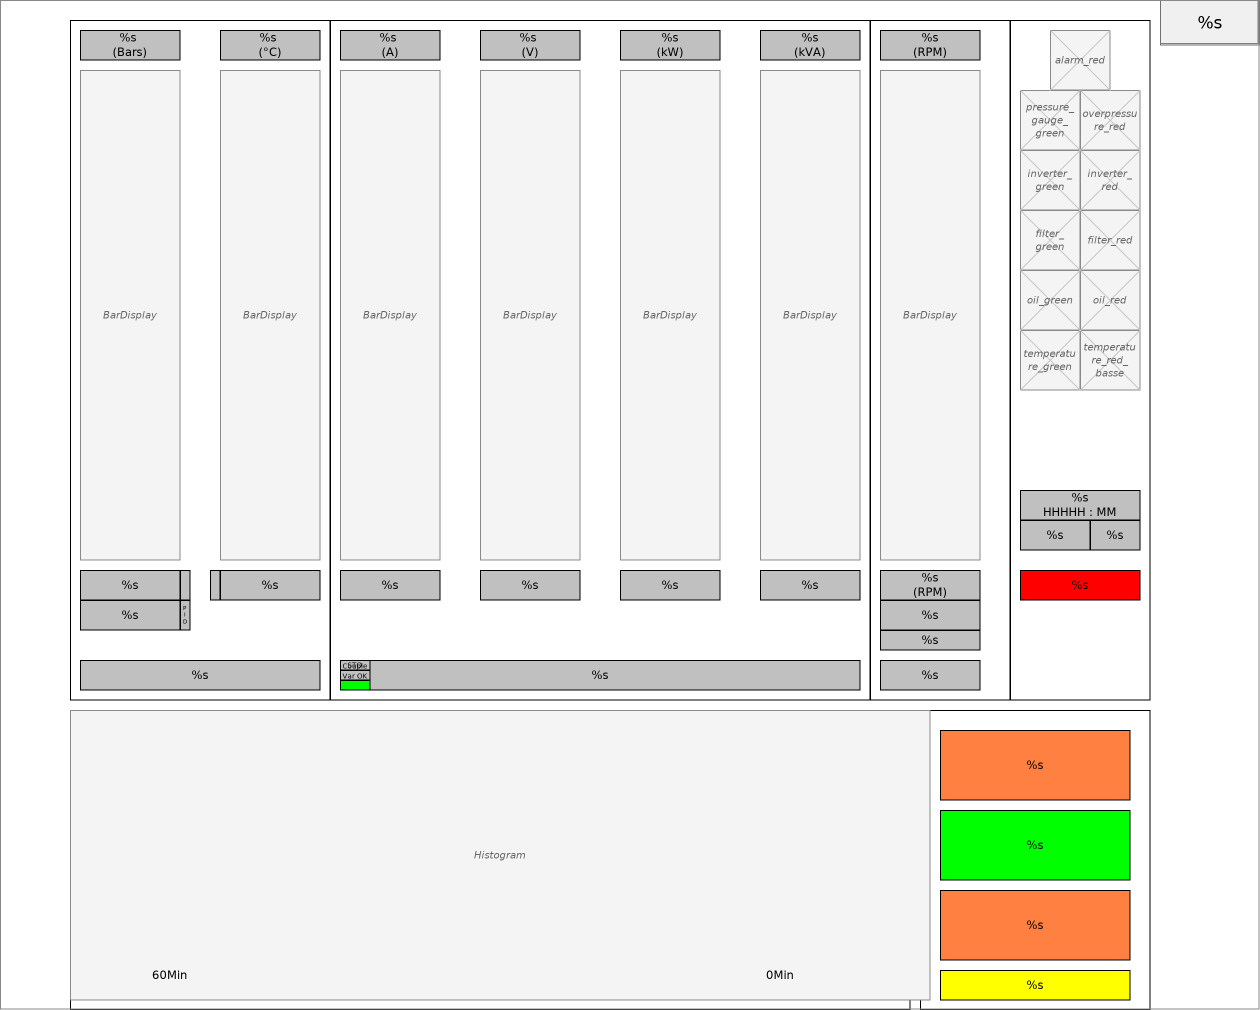
VISUALIZATION POMPE_ATOS_ECRAN  // 1260x1010, background image fond 19p 1280x1024
    Rectangle (70,710 840x300)
    Rectangle (1010,20 140x680)
    Rectangle (870,20 140x680)
    Rectangle (70,20 260x680), tooltip "Temperature huile"
    Rectangle (330,20 540x680)
    BarDisplay (80,70 100x490), value: Mesure_Pression, scale format: %.1f, scale 0..150
    BarDisplay (220,70 100x490), value: Mesure_Temperature_Huile, scale format: %.1f, scale 0..100
    Rectangle (80,570 100x30), "%s", text variable: Global_Atos.Mesure_Pression
    Rectangle (220,570 100x30), "%s", text variable: Mesure_Temperature_Huile
    Rectangle (80,30 100x30), "%s (Bars)", tooltip "Pression", text variable: Label[138]
    Rectangle (220,30 100x30), "%s (°C)", tooltip "Temperature huile", text variable: Label[83]
    BarDisplay (340,70 100x490), value: (INT_TO_LREAL(Lenze_Motor_Current_Motec_Pompe))/10, scale format: %.1f, scale 0..10
    Rectangle (340,570 100x30), "%s", text variable: (INT_TO_LREAL(Lenze_Motor_Current_Motec_Pompe))/10
    Rectangle (340,30 100x30), "%s (A)", tooltip "Courant", text variable: Label[139]
    BarDisplay (480,70 100x490), value: Lenze_Motor_Voltage_Var_Pompe, scale format: %.1f, scale 0..400
    Rectangle (480,570 100x30), "%s", text variable: Global_Atos.Lenze_Motor_Voltage_Var_Pompe
    Rectangle (480,30 100x30), "%s (V)", tooltip "Tension", text variable: Label[140]
    BarDisplay (620,70 100x490), value: (DINT_TO_LREAL(Lenze_Effective_Power_Var_Pompe))/1000, scale format: %.1f, scale 0..7
    Rectangle (620,570 100x30), "%s", text variable: (DINT_TO_LREAL(Lenze_Effective_Power_Var_Pompe))/1000
    Rectangle (620,30 100x30), "%s (kW)", tooltip "Puissance kW", text variable: Label[142]
    BarDisplay (760,70 100x490), value: (DINT_TO_LREAL (Lenze_Apparent_Power_Var_Pompe)/1000), scale format: %.1f, scale 0..7
    Rectangle (760,570 100x30), "%s", text variable: (DINT_TO_LREAL (Lenze_Apparent_Power_Var_Pompe)/1000)
    Rectangle (760,30 100x30), "%s (kVA)", tooltip "Puissance kVA", text variable: Label[142]
    Rectangle (80,660 240x30), "%s", tooltip "Pompe", text variable: Label[143]
    Rectangle (340,660 520x30), "%s", tooltip "Variateur Moteur", text variable: Label[144]
    BarDisplay (880,70 100x490), value: ABS(Lenze_Actual_Speed_Motec_Pompe), scale format: %.1f, scale 0..3200
    Rectangle (880,600 100x30), "%s", text variable: ABS(Lenze_Actual_Speed_Motec_Pompe)
    Rectangle (880,30 100x30), "%s (RPM)", tooltip "Vitesse ( RPM )", text variable: Label[141]
    Rectangle (880,570 100x30), "%s (RPM)", tooltip "Vitesse ( RPM)", text variable: Label[141]
    Rectangle (880,660 100x30), "%s", tooltip "Moteur", text variable: Label[145]
    Rectangle (1020,570 120x30), "%s", tooltip "Annulation defaut", text variable: Label[147], colour toggle: Global_Atos.Defaut_Centrale_Hydro
        tap Global_Atos.ACK_DEF
    Rectangle (430,960 100x30), "30Min", text variable: Global_Atos.Mesure_Pression
    Rectangle (1020,520 70x30), "%s", text variable: Global_Atos.NB_Heures_En_Service
    Rectangle (1090,520 50x30), "%s", text variable: Global_Atos.NB_Min_En_Service
    Rectangle (1020,490 120x30), "%s HHHHH : MM", tooltip "Temps", text variable: Label[146], colour toggle: (Defaut_Variateur) <> 0
    Rectangle (80,600 100x30), "%s", text variable: Global_Atos.Pression_Consigne_Temp
    Rectangle (920,710 230x300)
    Rectangle (940,970 190x30), "%s", tooltip "Mode de reglage", text variable: Label[152], colour toggle: Global_Atos.Mode_Reglage, invisible if: (Pompe_En_Service) <> 0
        toggle Global_Atos.Mode_Reglage
    Rectangle (940,730 190x70), "%s", tooltip "Augmenter Limiteur Pression", text variable: Label[149], invisible if: NOT Global_Atos.Limiteur_plus
    Rectangle (940,890 190x70), "%s", tooltip "Diminuer Limiteur Pression", text variable: Label[151], invisible if: NOT Global_Atos.Limiteur_moins
    Rectangle (940,810 190x70), "%s", tooltip "Pression OK", text variable: Label[150], invisible if: NOT Global_Atos.Pression_Reglage_OK
    Rectangle (880,630 100x20), "%s", text variable: TRUNC(ABS(PID_Out_RPM))
    Rectangle (180,570 10x30), colour toggle: Global_Atos.Pression_Ok
    Rectangle (210,570 10x30), colour toggle: NOT Global_Atos.Defaut_Temperature_Huile_Basse AND NOT Defaut_Temperature_Huile_Haute
    Rectangle (340,660 30x10), "STO", colour toggle: Global_Atos.Statut_STO_Pompe
    Rectangle (340,670 30x10), "Couple", colour toggle: Global_Atos.Statut_Sous_Couple_Pompe
    Rectangle (340,680 30x10), "Var OK", colour toggle: Global_Atos.Defaut_Variateur_Pompe
    Rectangle (180,600 10x30), "P I D", colour toggle: Global_Atos.PID_Actif
    Histogram (70,710 860x290), scale format: %.1f, scale -10..100
        p1518820177: TAB_Log_Before_Temperature_Fault
        p102497268: TAB_Log_Before_Temperature_Fault
        p788070771: ARRAY [0..60] OF INT
        p518627256: °C
    Image (1020,90 60x60), invisible if: (Defaut_Pression_Huile) <> 0, image: pressure_gauge_green
    Image (1080,90 60x60), invisible if: NOT Global_Atos.Defaut_Pression_Huile_Consigne, image: overpressure_red
    Image (1020,150 60x60), invisible if: Global_Atos.Defaut_Variateur_Pompe, image: inverter_green
    Image (1080,150 60x60), invisible if: NOT Global_Atos.Defaut_Variateur_Pompe, image: inverter_red
    Image (1020,210 60x60), invisible if: Global_Atos.Defaut_Filtre_Pompe, image: filter_green
    Image (1080,210 60x60), invisible if: NOT Global_Atos.Defaut_Filtre_Pompe, image: filter_red
    Image (1020,330 60x60), invisible if: (Global_Atos.Defaut_Temperature_Huile_Haute OR Defaut_Temperature_Huile_Basse OR Alarme_Temperature_Huile_Haute OR Alarme_Temperature_Huile_Basse) <> 0, image: temperature_green
    Image (1080,330 60x60), invisible if: NOT Global_Atos.Alarme_Temperature_Huile_Haute, image: temperature_orange
    Image (1080,330 60x60), invisible if: NOT Global_Atos.Alarme_Temperature_Huile_Basse, image: temperature_orange_basse
    Image (1050,30 60x60), invisible if: NOT Global_Atos.Defaut_Centrale_Hydro, image: alarm_red
    Image (1080,330 60x60), invisible if: NOT Global_Atos.Defaut_Temperature_Huile_Haute, image: temperature_red_haute
    Image (1080,330 60x60), invisible if: NOT Global_Atos.Defaut_Temperature_Huile_Basse, image: temperature_red_basse
    Image (1080,270 60x60), invisible if: NOT Global_Atos.Defaut_Niveau_Huile_Bas, image: oil_red
    Image (1020,270 60x60), invisible if: Global_Atos.Defaut_Niveau_Huile_Bas, image: oil_green
    Rectangle (730,960 100x30), "0Min", text variable: Global_Atos.Mesure_Pression
    Rectangle (120,960 100x30), "60Min", text variable: Global_Atos.Mesure_Pression
    Button (1160,0 100x45), "%s", text variable: Label[6]
        OnMouseUp: change screen: AssignExpression MenuPrincipal
END_VISUALIZATION

(* stored: Version 1.1.0.1
   Visu POMPE_ATOS_ECRAN: Id {d1b895a7-25b9-4866-8882-8d96d8537e3b} *)
